TEXTLIST HandlingModulesState
  10 = 'Stop Run'
  19 = 'Stop End'
  20 = 'Reset Run'
  21 = 'Reset End'
  60 = 'Power Run'
  69 = 'Power End'
  100 = 'Home Run'
  109 = 'Home End'
  300 = 'Man Run'
  399 = 'Man End'
  500 = 'Load Run'
  599 = 'Load End'
  3000 = 'Move Run'
  3099 = 'Move End'
  800 = 'Unload Run'
  899 = 'Unload End'
  1000 = 'Do Run'
  1099 = 'Do End'
  1 = ''
   = ''
END_TEXTLIST

(* stored: Version 1.1.0.1, ProductVersion 3.1.4024.11
   TextList HandlingModulesState: Id {f1f070d4-b623-4808-b34a-ebacbab00682} *)
